{attribute 'no_explicit_call' := 'DriectOnlineStarterMotor is a CLASS and must be accessed using methods or properties'}
FUNCTION_BLOCK DirectOnlineStarterMotor implements I_SingleDirectionMotor
VAR
	contactor			: Contactor;
END_VAR

METHOD Start
contactor.SwitchOn();
END_METHOD

METHOD Stop
contactor.SwitchOff();
END_METHOD

END_FUNCTION_BLOCK

(* stored: Version 1.1.0.1, ProductVersion 3.1.4024.11
   POU DirectOnlineStarterMotor: Id {a101c44b-39dc-47a0-aa83-2f5e8d3ebc8f}, SpecialFunc None
   Method Start: Id {a4e06773-ad0e-4233-b123-7fe84f394d3b}
   Method Stop: Id {039e0f25-4076-41f4-ae24-9d552466c094} *)
